// TIA Portal V21 export
TYPE "motorInterface"
   STRUCT
      status : "motorStatus";
      statusWord { S7_SetPoint := 'True'} : Word;
      "step" : USInt;
      stepTime : LTime;
      speedSp : Real;
      speedPv : Real;
      alm { S7_SetPoint := 'True'} : "motorAlm";   // active alarms
      almWord { S7_SetPoint := 'True'} : Word;
      stopCtx { S7_SetPoint := 'True'} : "motorStopCtx";
   END_STRUCT;
END_TYPE
